PROGRAM P92_Maintenance
VAR
	(* Input *)
	//Light
	rTrigReactorCabinetSwitch	: R_TRIG;
	rTrigReactorCabinetMagnet 	: R_TRIG;
	fTrigReactorCabinetMagnet 	: F_TRIG;
	rTrigGasCabinetSwitch		: R_TRIG;
	rTrigGasCabinetMagnet		: R_TRIG;
	fTrigGasCabinetMagnet		: F_TRIG;

	bReactorCabinetLampSwitch : BOOL;
	bGasCabinetLampSwitch	: BOOL;
	
	bReactorCabientMagnet	: BOOL;
	bGasCabinetMagnet		: BOOL;
	bPowerDistributeMagnet	: BOOL;
	
	(* Output to Device *)
	// Cabinet Lamp
	bReactorCabinetLamp		: BOOL;
	bGasCabinetLamp			: BOOL;
	bPowerDistributeLamp	: BOOL;
	
	bSMPS24V480WFault		: BOOL;
	bSMPS24V72WFault		: BOOL;
	bSMPS15VPlusFault		: BOOL;
	bSMPS15VMinusFault		: BOOL;
	// Signal Tower
	bSignalTower			: BYTE;
	TimerSignalTower		: TON;
	bBuzzer					: BOOL;
END_VAR

(* Read from Device Value *)
//Lamp
bReactorCabientMagnet 	:= GVL_IO_REACTOR_CABINET.DI_03_ReactorCabinetDoorClose;
bGasCabinetMagnet 		:= GVL_IO_GAS_CABINET.DI_01_GasCabinetDoorClose;
bPowerDistributeMagnet	:= GVL_IO_GAS_CABINET.DI_01_ControlCabinetDoorClose;

//SMPS
bSMPS24V480WFault	:= NOT(GVL_IO_GAS_CABINET.DI_01_SMPS_1Alarm);
bSMPS24V72WFault	:= NOT(GVL_IO_GAS_CABINET.DI_01_SMPS_2Alarm);
bSMPS15VPlusFault	:= NOT(GVL_IO_GAS_CABINET.DI_01_SMPS_3Alarm);
bSMPS15VMinusFault	:= NOT(GVL_IO_GAS_CABINET.DI_02_SMPS_4Alarm);


// Reactor Cabinet Lamp
rTrigReactorCabinetSwitch(CLK:=GVL_IO_REACTOR_CABINET.DI_01_ReactorCabinetLampButton);
fTrigReactorCabinetMagnet(CLK:=GVL_IO_REACTOR_CABINET.DI_03_ReactorCabinetDoorClose);

IF rTrigReactorCabinetSwitch.Q OR rTrigReactorCabinetMagnet.Q OR fTrigReactorCabinetMagnet.Q THEN
	bReactorCabinetLamp := NOT(bReactorCabinetLamp);
END_IF
// Gas Delivery Cabinet Lamp
rTrigGasCabinetSwitch(CLK:= GVL_IO_GAS_CABINET.DI_01_GasCabinetLampButton);
rTrigGasCabinetMagnet(CLK:= GVL_IO_GAS_CABINET.DI_01_GasCabinetDoorClose);

IF rTrigGasCabinetSwitch.Q THEN
	bGasCabinetLamp := NOT(bGasCabinetLamp);
ELSIF fTrigGasCabinetMagnet.Q THEN
	bGasCabinetLamp := TRUE;
ELSIF rTrigGasCabinetMagnet.Q THEN
	bGasCabinetLamp := FALSE;
END_IF
// Power Distribute Unit Lamp
bPowerDistributeLamp := NOT(bPowerDistributeMagnet); //Magnet Switch

(* Buzzer On/Off *)
IF bBuzzer <> GVL_IO.aInterlockEnable[1].2 THEN
	bBuzzer := GVL_IO.aInterlockEnable[1].2;
END_IF

(* Blink Signal Tower *)
CASE GVL_IO.nCaseSignalTower OF
	1: //RED 
		TimerSignalTower(IN:=TRUE, PT:=T#500MS);
		IF TimerSignalTower.Q THEN
			TimerSignalTower(IN:=FALSE);
			IF bSignalTower = 0 THEN
				bSignalTower := 2#0000_0001; // RED
			ELSE
				bSignalTower := 0;
			END_IF
		END_IF

	2: //YELLOW 
		TimerSignalTower(IN:=TRUE, PT:=T#1S);
		IF TimerSignalTower.Q THEN
			TimerSignalTower(IN:=FALSE);
			IF bSignalTower = 0 THEN
				bSignalTower := 2#0000_0010; // YELLOW
			ELSE
				bSignalTower := 0;
			END_IF
		END_IF
	3: //GREEN
		TimerSignalTower(IN:=TRUE, PT:=T#1S);
		IF TimerSignalTower.Q THEN
			TimerSignalTower(IN:=FALSE);
			IF bSignalTower = 0 THEN
				bSignalTower := 2#0000_0100; // GREEN
			ELSE
				bSignalTower := 0;
			END_IF
		END_IF
	4: //BLUE
		bSignalTower := 2#0000_1000;
	5: //WHITE
		bSignalTower := 2#0001_0000;
END_CASE

(* Write to Device Value *)
GVL_IO_REACTOR_CABINET.DO_06_ReactorCabinetLamp := bReactorCabinetLamp;
GVL_IO_GAS_CABINET.DO_07_GasCabinetLamp := bGasCabinetLamp;
GVL_IO_GAS_CABINET.DO_07_ControlCabinetLamp := bPowerDistributeLamp;


GVL_IO_REACTOR_CABINET.DO_04_SignalTowerRed:=bSignalTower.0; //0:RED-Alarm,
GVL_IO_REACTOR_CABINET.DO_04_SignalTowerOrange:=bSignalTower.1; //1:YELLOW,-Warning
GVL_IO_REACTOR_CABINET.DO_04_SignalTowerGreen:=bSignalTower.2; //2:GREEN-Running
GVL_IO_REACTOR_CABINET.DO_04_SignalTowerBlue:=bSignalTower.3; //3:BLUE-Idle
GVL_IO_REACTOR_CABINET.DO_04_SignalTowerWhite:=bSignalTower.4; //4:WHITE-Maint
GVL_IO_REACTOR_CABINET.DO_04_SignalTowerBuzzer:=bBuzzer; //5:BUZZER-Alarm


////SignalTower
//GVL_IO.aDigitalOutputIO[1].0 	:= bSignalTower.0; //0:RED-Alarm,
//GVL_IO.aDigitalOutputIO[1].1 	:= bSignalTower.1; //1:YELLOW,-Warning 
//GVL_IO.aDigitalOutputIO[1].2 	:= bSignalTower.2; //2:GREEN-Running
//GVL_IO.aDigitalOutputIO[1].3 	:= bSignalTower.3; //3:BLUE-Idle
//GVL_IO.aDigitalOutputIO[1].4 	:= bSignalTower.4; //4:WHITE-Maint
//GVL_IO.aDigitalOutputIO[1].5 	:= bBuzzer; //5:BUZZER-Alarm

END_PROGRAM

(* stored: Version 1.1.0.1, ProductVersion 3.1.4024.15
   POU P92_Maintenance: Id {17478ea4-373a-4676-aa4e-f86e85a19514}, SpecialFunc None *)
